TYPE PrintingStates :
(	
	PrepareModel,
	SlicePrint,
	Print,
	FinishPrint
	) := PrepareModel;
END_TYPE

(* stored: Version 1.1.0.1, ProductVersion 3.1.4024.15
   DUT PrintingStates: Id {e41d79aa-1416-46b8-b40c-53a0261f0449} *)
